(* CoDeSys 2.3 export: PLC_PRG.EXP *)

(* POU PLC_PRG, ST *)
PROGRAM PLC_PRG
VAR
	p, p1: POINTER TO BYTE;
	pip: POINTER TO IPAddress;
	parr: POINTER TO ARRAY [0..3] OF INT;
	N: INT:= 6;
	arrInit: BOOL;
	i: INT;
END_VAR
IF NOT arrInit THEN
	p:= NewArray(10, 2);
	arrInit:= TRUE;
END_IF;

	pip:= p;
	(*p1:= p+3;
	p1^:= 1;
	i:= parr^[1];*)
	FOR i := 0 TO pip^.length - 1 DO
		pip^.items[i] := 1;
	END_FOR;
END_PROGRAM
